TYPE Basic_MC_MoveVelocity_Status_typ : 	
	STRUCT 
		In_Velocity : BOOL;
		Busy : BOOL;
		CommandAborted : BOOL;
		Active : BOOL ;
	END_STRUCT
END_TYPE

(* stored: Version 1.1.0.1, ProductVersion 3.1.4024.3
   DUT Basic_MC_MoveVelocity_Status_typ: Id {886b36ef-ff4d-05f6-3316-784534e2f9d3} *)
